(* Schneider Machine Expert - Basic project H_DUSTER, file version 2.9.0.0 *)
(* CompanyInformations: Name=PROMASS, PhoneNumber=+39074238501, Street=Via XXV Aprile, 10/12, City=Trevi, ZipCode=06039, State=PG, Country=Italy, WebSite=www.promass.com *)
(* ProjectInformations: Name=MIXER_EPP, Description=CONTROL TO MIX-UP RECYCLED EPP (EXANDED POLYPROPILENE) WITH FRESH EPP.
AN ADDITIONAL BLOWE IS ADDED TO PERMIT THE OUTPUT FLOW *)
(* UserInformations: LastName=Torroni, FirstName=Stefano, PhoneNumber=+390742385051, Email=info@promass.com, Street=via XXV Aprile, 10/12, City=Trevi, ZipCode=06039, State=Umbria, Country=Italy *)

HARDWARE
  Cpu 0: TM221CE16T
  EthernetConfiguration: NetworkName=M221, IpAllocationMode=FixedAddress, IpAddress=192.168.250.10, SubnetMask=255.255.255.0
  SerialLineConfiguration: Baud=Baud19200, Parity=ParityEven, DataBits=DataBits8, StopBits=StopBits1, PhysicalMedium=PhysicalMediumRs485, TransmissionMode=TransmissionModeIoScannerRtu
  MastTask: UsePeriodScanMode=false, PeriodScan=100
  FastTask: Period=255
  CpuBehavior: StartingMode=StartAutoRunForced, AutoSaveRamOnEeprom=true, WatchdogPeriod=250

SYMBOLS  (address, symbol, comment, settings)
  %M0       DRV_PWR_ON
  %M1       DRV1_JOG_INC
  %M2       DRV1_JOG_DEC
  %M3       DRV2_JOG_INC
  %M4       DRV2_JOG_DEC
  %M5       DRV1_MOVE_VEL
  %M6       DRV2_MOVE_VEL
  %M7       DRV1_ERROR
  %M8       DRV2_ERROR
  %M11      UPP_SENS_ON
  %M12      REM_TANK_FULL_V
  %M13      BLOWER_TOF
  %M20      DRV3_JOG_INC
  %M21      DRV3_JOG_DEC
  %M22      DRV4_JOG_INC
  %M23      DRV4_JOG_DEC
  %M24      DRV3_MOVE_VEL
  %M25      DRV4_MOVE_VEL
  %M26      DRV3_ERROR
  %M27      DRV4_ERROR
  %M30      U1_POWER_ON
  %M31      U2_POWER_ON
  %M32      U3_POWER_ON
  %M33      U4_POWER_ON
  %M34      U1_DRIVE_ERR
  %M35      U2_DRIVE_ERR
  %M36      U3_DRIVE_ERR
  %M37      U4_DRIVE_ERR
  %M40      DRV1_CONTMOTION
  %M41      DRV2_CONTMOTION
  %M42      DRV3_CONTMOTION
  %M43      DRV4_CONTMOTION
  %M100     RATIO_0_CHANGED
  %M101     RATIO_1_CHANGED
  %MW0      DRV1_JOG_SPEED
  %MW1      DRV2_JOG_SPEED
  %MW2      DRV1_MOVEVEL_SPEED
  %MW3      DRV2_MOVE_VEL_SPEED
  %MW4      HMI_ALARMS
  %MW5      FSM
  %MW6      HMI_INP_00  "HMI>>PLC COMMANDS WORD 01"
  %MW7      HMI_OUT_00  "PLC>>HMI FEEDBACK WORD 01"
  %MW8      HMI_OUT_01  "PLC>>HMI FEEDBACK WORD 02"
  %MW9      U1_M1_SPEED_RPM_OUT
  %MW10     U2_M2_SPEED_RPM_OUT
  %MW11     U3_M3_SPEED_RPM_OUT
  %MW12     U4_M4_SPEED_RPM_OUT
  %MW14     DRV3_JOG_SPEED
  %MW15     DRV4_JOG_SPEED
  %MW16     DRV3_MOVEVEL_SPEED
  %MW17     DRV4_MOVEVEL_SPEED
  %MW18     U1_M1_GEARBOX_RATIO  "RECYCLED_MATERIAL SCREW GEARBOX => i=15"
  %MW19     U2_M2_GEARBOX_RATIO  "STAR VALVE INLET GEARBOX => i=120"
  %MW20     U3_M3_GEARBOX_RATIO  "STAR VALVE OUTLET GEARBOX => i=40"
  %MW21     U4_M4_GEARBOX_RATIO  "FAN BLOWER DOES NOT HAVE GEARBOX => i=1"
  %MW22     HMI_INP_02  "HMI>>PLC COMMANDS WORD 02"
  %MW24     HMI_OUT_02  "PLC>>HMI FEEDBACK WORD 03"
  %MW25     FSM_FEEDBACK
  %MW30     DRV1_SPD_AUTO  "RECYCLING MATERIAL DRIVE SPEED AUTOMODE (MULTIPLY BY 2.58 DUE TO GEAR RATIO 12.4/4.8 <=>GEAR_RATIO0/GEAR_RATIO1"
  %MW31     DRV2_SPD_AUTO  "RAW MATERIAL DRIVE SPEED AUTOMODE"
  %MW32     DRV1_SPD_AUTO0
  %MW33     DRV2_SPD_AUTO0
  %MW34     DRV3_SPD_AUTO
  %MW35     DRV4_SPD_AUTO
  %MW36     DRV3_SPD_AUTO0
  %MW37     DRV4_SPD_AUTO0
  %MC_JOG_ATV0   [Axis(Value(DriveAxis=DRV0)), Vel(Value(short=210))]
  %MC_JOG_ATV1   [Axis(Value(DriveAxis=DRV1)), Vel(Value(short=210))]
  %MC_JOG_ATV2   [Axis(Value(DriveAxis=DRV2)), Vel(Value(short=210))]
  %MC_JOG_ATV3   [Axis(Value(DriveAxis=DRV3)), Vel(Value(short=400))]
  %MC_MOVEVEL_ATV0   [Axis(Value(DriveAxis=DRV0)), Vel(Value(short=0))]
  %MC_MOVEVEL_ATV1   [Axis(Value(DriveAxis=DRV1)), Vel(Value(short=0))]
  %MC_MOVEVEL_ATV2   [Axis(Value(DriveAxis=DRV2)), Vel(Value(short=0))]
  %MC_MOVEVEL_ATV3   [Axis(Value(DriveAxis=DRV3)), Vel(Value(short=0))]
  %MC_POWER_ATV0   [Axis(Value(DriveAxis=DRV0))]
  %MC_POWER_ATV1   [Axis(Value(DriveAxis=DRV1))]
  %MC_POWER_ATV2   [Axis(Value(DriveAxis=DRV2))]
  %MC_POWER_ATV3   [Axis(Value(DriveAxis=DRV3))]
  %MC_READMOTIONSTATE_ATV0   [Axis(Value(DriveAxis=DRV0))]
  %MC_READMOTIONSTATE_ATV1   [Axis(Value(DriveAxis=DRV1))]
  %MC_READMOTIONSTATE_ATV2   [Axis(Value(DriveAxis=DRV2))]
  %MC_READMOTIONSTATE_ATV3   [Axis(Value(DriveAxis=DRV3))]
  %MC_READSTATUS_ATV0   [Axis(Value(DriveAxis=DRV0))]
  %MC_READSTATUS_ATV1   [Axis(Value(DriveAxis=DRV1))]
  %MC_READSTATUS_ATV2   [Axis(Value(DriveAxis=DRV2))]
  %MC_READSTATUS_ATV3   [Axis(Value(DriveAxis=DRV3))]
  %MC_RESET_ATV0   [Axis(Value(DriveAxis=DRV0))]
  %MC_RESET_ATV1   [Axis(Value(DriveAxis=DRV1))]
  %MC_RESET_ATV2   [Axis(Value(DriveAxis=DRV2))]
  %MC_RESET_ATV3   [Axis(Value(DriveAxis=DRV3))]
  %MC_STOP_ATV0   [Axis(Value(DriveAxis=DRV0))]
  %MC_STOP_ATV1   [Axis(Value(DriveAxis=DRV1))]
  %MC_STOP_ATV2   [Axis(Value(DriveAxis=DRV2))]
  %MC_STOP_ATV3   [Axis(Value(DriveAxis=DRV3))]
  %I0.0     START_BTN
  %I0.1     STOP_BTN
  %I0.2     QM1
  %I0.3     QM2
  %I0.4     QM3
  %I0.5     QM4
  %Q0.0     STO
  %Q0.1     KA2_MILL_01_IF
  %Q0.2     KA3_MILL_02_IF

POU MAIN
  (* SectionNumber=1 *)

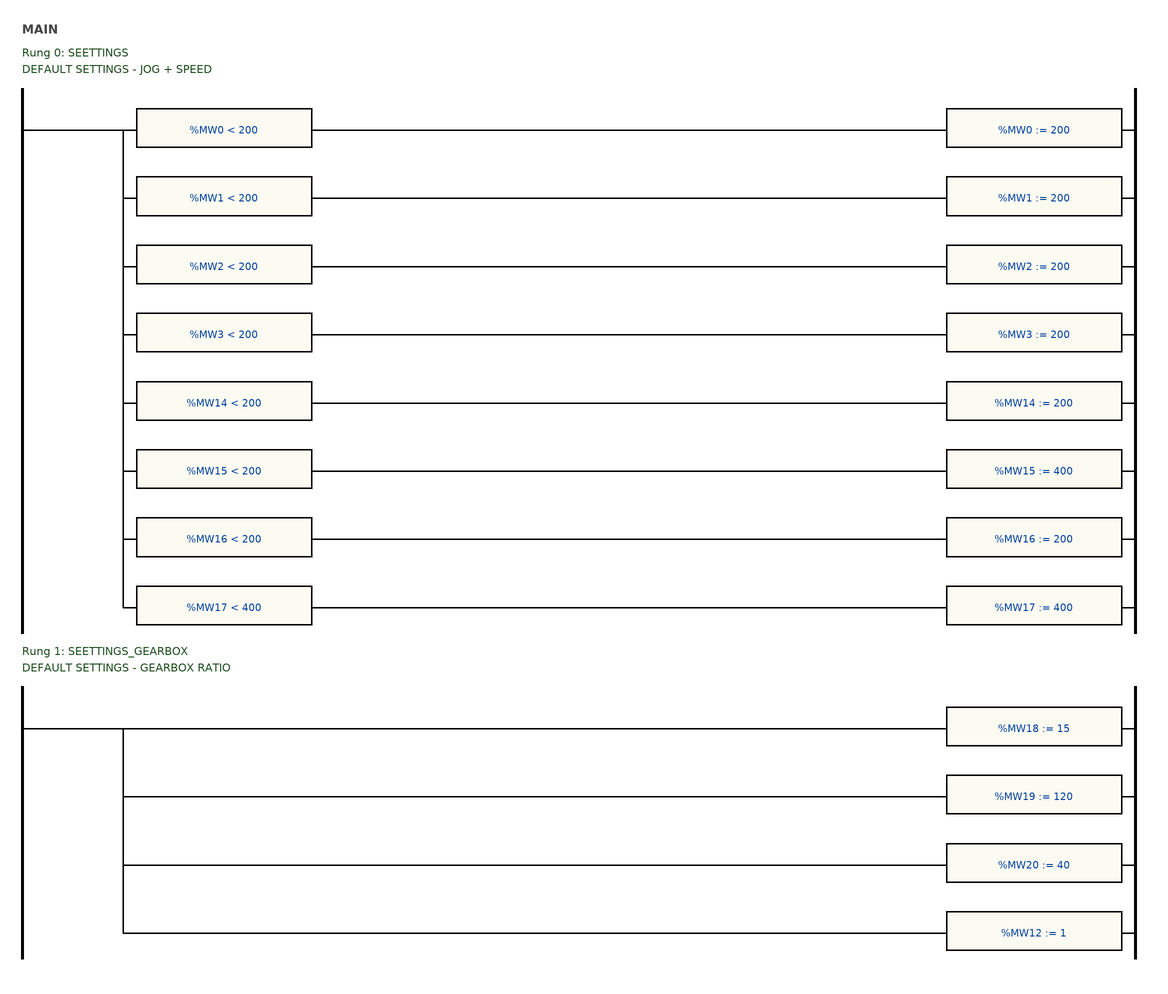

// Rung 0: SEETTINGS
// DEFAULT SETTINGS - JOG + SPEED
  LD 1
  MPS
  AND [ %MW0 < 200 ]      (* DRV1_JOG_SPEED *)
  [ %MW0 := 200 ]         (* DRV1_JOG_SPEED *)
  MRD
  AND [ %MW1 < 200 ]      (* DRV2_JOG_SPEED *)
  [ %MW1 := 200 ]         (* DRV2_JOG_SPEED *)
  MRD
  AND [ %MW2 < 200 ]      (* DRV1_MOVEVEL_SPEED *)
  [ %MW2 := 200 ]         (* DRV1_MOVEVEL_SPEED *)
  MRD
  AND [ %MW3 < 200 ]      (* DRV2_MOVE_VEL_SPEED *)
  [ %MW3 := 200 ]         (* DRV2_MOVE_VEL_SPEED *)
  MRD
  AND [ %MW14 < 200 ]     (* DRV3_JOG_SPEED *)
  [ %MW14 := 200 ]        (* DRV3_JOG_SPEED *)
  MRD
  AND [ %MW15 < 200 ]     (* DRV4_JOG_SPEED *)
  [ %MW15 := 400 ]        (* DRV4_JOG_SPEED *)
  MRD
  AND [ %MW16 < 200 ]     (* DRV3_MOVEVEL_SPEED *)
  [ %MW16 := 200 ]        (* DRV3_MOVEVEL_SPEED *)
  MPP
  AND [ %MW17 < 400 ]     (* DRV4_MOVEVEL_SPEED *)
  [ %MW17 := 400 ]        (* DRV4_MOVEVEL_SPEED *)
  // as ST:
  //   IF DRV1_JOG_SPEED < 200 THEN DRV1_JOG_SPEED := 200; END_IF;
  //   IF DRV2_JOG_SPEED < 200 THEN DRV2_JOG_SPEED := 200; END_IF;
  //   IF DRV1_MOVEVEL_SPEED < 200 THEN DRV1_MOVEVEL_SPEED := 200; END_IF;
  //   IF DRV2_MOVE_VEL_SPEED < 200 THEN DRV2_MOVE_VEL_SPEED := 200; END_IF;
  //   IF DRV3_JOG_SPEED < 200 THEN DRV3_JOG_SPEED := 200; END_IF;
  //   IF DRV4_JOG_SPEED < 200 THEN DRV4_JOG_SPEED := 400; END_IF;
  //   IF DRV3_MOVEVEL_SPEED < 200 THEN DRV3_MOVEVEL_SPEED := 200; END_IF;
  //   IF DRV4_MOVEVEL_SPEED < 400 THEN DRV4_MOVEVEL_SPEED := 400; END_IF;

// Rung 1: SEETTINGS_GEARBOX
// DEFAULT SETTINGS - GEARBOX RATIO
  LD 1
  [ %MW18 := 15 ]         (* U1_M1_GEARBOX_RATIO *)
  [ %MW19 := 120 ]        (* U2_M2_GEARBOX_RATIO *)
  [ %MW20 := 40 ]         (* U3_M3_GEARBOX_RATIO *)
  [ %MW12 := 1 ]          (* U4_M4_SPEED_RPM_OUT *)
  // as ST:
  //   U1_M1_GEARBOX_RATIO := 15;
  //   U2_M2_GEARBOX_RATIO := 120;
  //   U3_M3_GEARBOX_RATIO := 40;
  //   U4_M4_SPEED_RPM_OUT := 1;

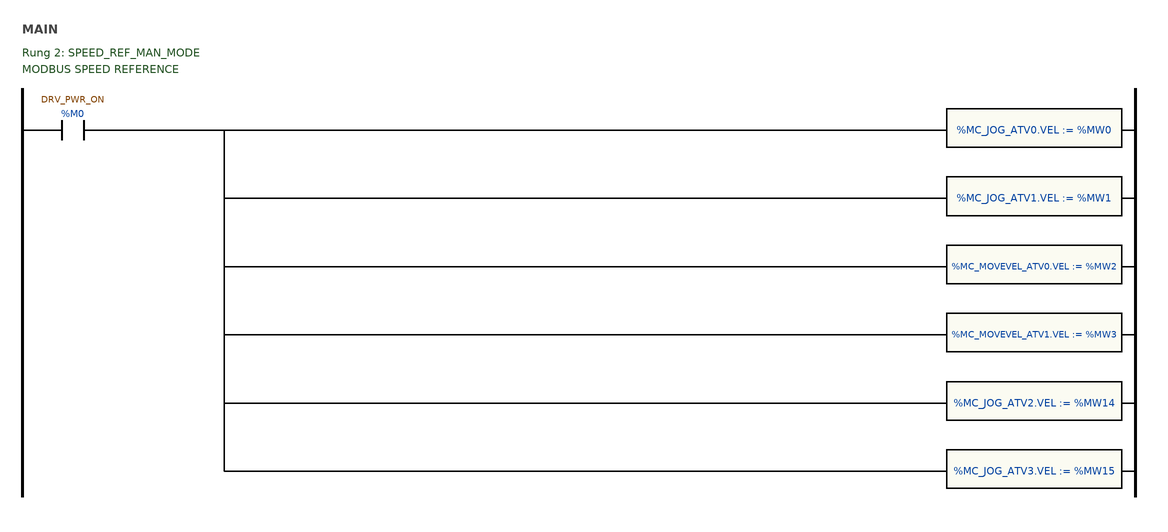

// Rung 2: SPEED_REF_MAN_MODE
// MODBUS SPEED REFERENCE
  LD %M0                  (* DRV_PWR_ON *)
  [ %MC_JOG_ATV0.VEL := %MW0 ](* DRV1_JOG_SPEED *)
  [ %MC_JOG_ATV1.VEL := %MW1 ](* DRV2_JOG_SPEED *)
  [ %MC_MOVEVEL_ATV0.VEL := %MW2 ](* DRV1_MOVEVEL_SPEED *)
  [ %MC_MOVEVEL_ATV1.VEL := %MW3 ](* DRV2_MOVE_VEL_SPEED *)
  [ %MC_JOG_ATV2.VEL := %MW14 ](* DRV3_JOG_SPEED *)
  [ %MC_JOG_ATV3.VEL := %MW15 ](* DRV4_JOG_SPEED *)
  // as ST:
  //   IF DRV_PWR_ON THEN %MC_JOG_ATV0.VEL := DRV1_JOG_SPEED; END_IF;
  //   IF DRV_PWR_ON THEN %MC_JOG_ATV1.VEL := DRV2_JOG_SPEED; END_IF;
  //   IF DRV_PWR_ON THEN %MC_MOVEVEL_ATV0.VEL := DRV1_MOVEVEL_SPEED; END_IF;
  //   IF DRV_PWR_ON THEN %MC_MOVEVEL_ATV1.VEL := DRV2_MOVE_VEL_SPEED; END_IF;
  //   IF DRV_PWR_ON THEN %MC_JOG_ATV2.VEL := DRV3_JOG_SPEED; END_IF;
  //   IF DRV_PWR_ON THEN %MC_JOG_ATV3.VEL := DRV4_JOG_SPEED; END_IF;

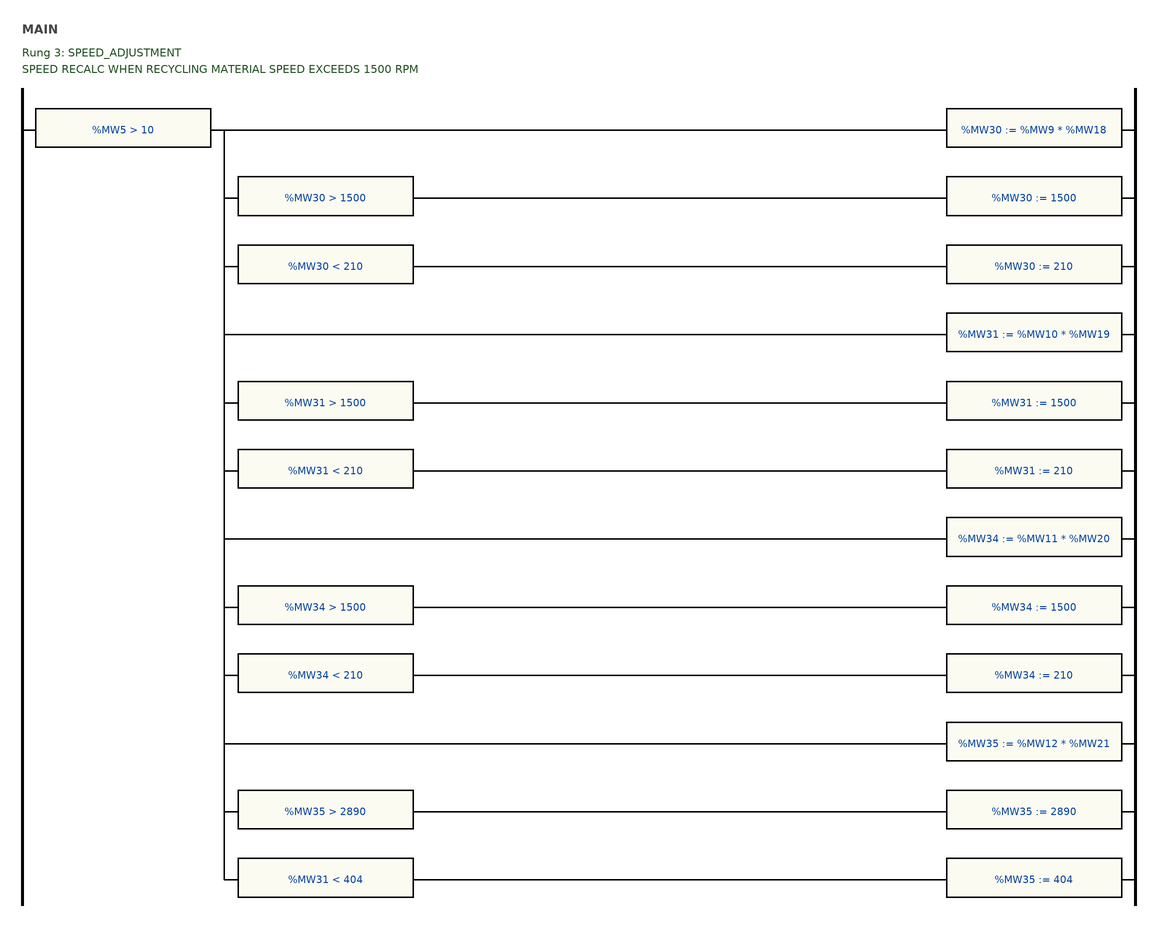

// Rung 3: SPEED_ADJUSTMENT
// SPEED RECALC WHEN RECYCLING MATERIAL SPEED EXCEEDS 1500 RPM
  LD [ %MW5 > 10 ]        (* FSM *)
  MPS
  [ %MW30 := %MW9 * %MW18 ](* DRV1_SPD_AUTO, U1_M1_SPEED_RPM_OUT, U1_M1_GEARBOX_RATIO *)
  MRD
  AND [ %MW30 > 1500 ]    (* DRV1_SPD_AUTO *)
  [ %MW30 := 1500 ]       (* DRV1_SPD_AUTO *)
  MRD
  AND [ %MW30 < 210 ]     (* DRV1_SPD_AUTO *)
  [ %MW30 := 210 ]        (* DRV1_SPD_AUTO *)
  MRD
  [ %MW31 := %MW10 * %MW19 ](* DRV2_SPD_AUTO, U2_M2_SPEED_RPM_OUT, U2_M2_GEARBOX_RATIO *)
  MRD
  AND [ %MW31 > 1500 ]    (* DRV2_SPD_AUTO *)
  [ %MW31 := 1500 ]       (* DRV2_SPD_AUTO *)
  MRD
  AND [ %MW31 < 210 ]     (* DRV2_SPD_AUTO *)
  [ %MW31 := 210 ]        (* DRV2_SPD_AUTO *)
  MRD
  [ %MW34 := %MW11 * %MW20 ](* DRV3_SPD_AUTO, U3_M3_SPEED_RPM_OUT, U3_M3_GEARBOX_RATIO *)
  MRD
  AND [ %MW34 > 1500 ]    (* DRV3_SPD_AUTO *)
  [ %MW34 := 1500 ]       (* DRV3_SPD_AUTO *)
  MRD
  AND [ %MW34 < 210 ]     (* DRV3_SPD_AUTO *)
  [ %MW34 := 210 ]        (* DRV3_SPD_AUTO *)
  MRD
  [ %MW35 := %MW12 * %MW21 ](* DRV4_SPD_AUTO, U4_M4_SPEED_RPM_OUT, U4_M4_GEARBOX_RATIO *)
  MRD
  AND [ %MW35 > 2890 ]    (* DRV4_SPD_AUTO *)
  [ %MW35 := 2890 ]       (* DRV4_SPD_AUTO *)
  MPP
  AND [ %MW31 < 404 ]     (* DRV2_SPD_AUTO *)
  [ %MW35 := 404 ]        (* DRV4_SPD_AUTO *)
  // as ST:
  //   IF FSM > 10 THEN DRV1_SPD_AUTO := U1_M1_SPEED_RPM_OUT * U1_M1_GEARBOX_RATIO; END_IF;
  //   IF FSM > 10 AND DRV1_SPD_AUTO > 1500 THEN DRV1_SPD_AUTO := 1500; END_IF;
  //   IF FSM > 10 AND DRV1_SPD_AUTO < 210 THEN DRV1_SPD_AUTO := 210; END_IF;
  //   IF FSM > 10 THEN DRV2_SPD_AUTO := U2_M2_SPEED_RPM_OUT * U2_M2_GEARBOX_RATIO; END_IF;
  //   IF FSM > 10 AND DRV2_SPD_AUTO > 1500 THEN DRV2_SPD_AUTO := 1500; END_IF;
  //   IF FSM > 10 AND DRV2_SPD_AUTO < 210 THEN DRV2_SPD_AUTO := 210; END_IF;
  //   IF FSM > 10 THEN DRV3_SPD_AUTO := U3_M3_SPEED_RPM_OUT * U3_M3_GEARBOX_RATIO; END_IF;
  //   IF FSM > 10 AND DRV3_SPD_AUTO > 1500 THEN DRV3_SPD_AUTO := 1500; END_IF;
  //   IF FSM > 10 AND DRV3_SPD_AUTO < 210 THEN DRV3_SPD_AUTO := 210; END_IF;
  //   IF FSM > 10 THEN DRV4_SPD_AUTO := U4_M4_SPEED_RPM_OUT * U4_M4_GEARBOX_RATIO; END_IF;
  //   IF FSM > 10 AND DRV4_SPD_AUTO > 2890 THEN DRV4_SPD_AUTO := 2890; END_IF;
  //   IF FSM > 10 AND DRV2_SPD_AUTO < 404 THEN DRV4_SPD_AUTO := 404; END_IF;

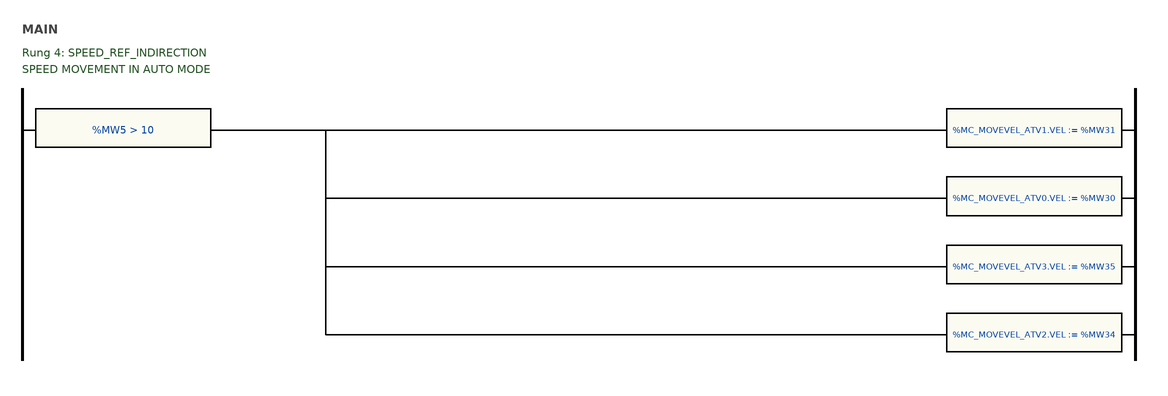

// Rung 4: SPEED_REF_INDIRECTION
// SPEED MOVEMENT IN AUTO MODE
  LD [ %MW5 > 10 ]        (* FSM *)
  [ %MC_MOVEVEL_ATV1.VEL := %MW31 ](* DRV2_SPD_AUTO *)
  [ %MC_MOVEVEL_ATV0.VEL := %MW30 ](* DRV1_SPD_AUTO *)
  [ %MC_MOVEVEL_ATV3.VEL := %MW35 ](* DRV4_SPD_AUTO *)
  [ %MC_MOVEVEL_ATV2.VEL := %MW34 ](* DRV3_SPD_AUTO *)
  // as ST:
  //   IF FSM > 10 THEN %MC_MOVEVEL_ATV1.VEL := DRV2_SPD_AUTO; END_IF;
  //   IF FSM > 10 THEN %MC_MOVEVEL_ATV0.VEL := DRV1_SPD_AUTO; END_IF;
  //   IF FSM > 10 THEN %MC_MOVEVEL_ATV3.VEL := DRV4_SPD_AUTO; END_IF;
  //   IF FSM > 10 THEN %MC_MOVEVEL_ATV2.VEL := DRV3_SPD_AUTO; END_IF;

POU FSM+CMD+HMI
  (* SectionNumber=2 *)

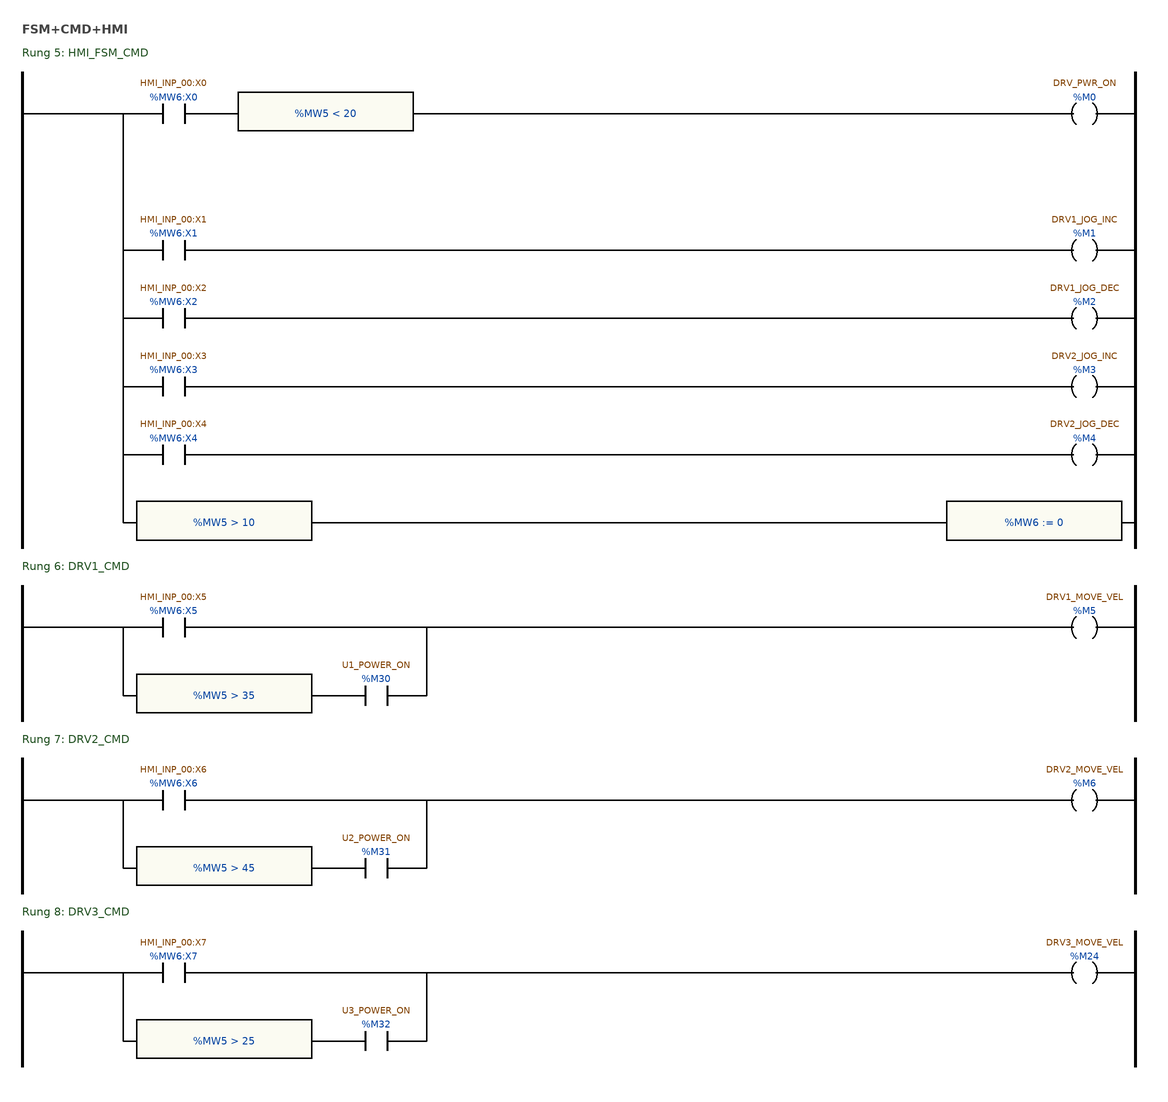

// Rung 5: HMI_FSM_CMD
  LD 1
  MPS
  AND %MW6:X0             (* HMI_INP_00 *)
  AND [ %MW5 < 20 ]       (* FSM *)
  ST %M0                  (* DRV_PWR_ON *)
  MRD
  AND %MW6:X1             (* HMI_INP_00 *)
  ST %M1                  (* DRV1_JOG_INC *)
  MRD
  AND %MW6:X2             (* HMI_INP_00 *)
  ST %M2                  (* DRV1_JOG_DEC *)
  MRD
  AND %MW6:X3             (* HMI_INP_00 *)
  ST %M3                  (* DRV2_JOG_INC *)
  MRD
  AND %MW6:X4             (* HMI_INP_00 *)
  ST %M4                  (* DRV2_JOG_DEC *)
  MPP
  AND [ %MW5 > 10 ]       (* FSM *)
  [ %MW6 := 0 ]           (* HMI_INP_00 *)
  // as ST:
  //   DRV_PWR_ON := HMI_INP_00:X0 AND FSM < 20;
  //   DRV1_JOG_INC := HMI_INP_00:X1;
  //   DRV1_JOG_DEC := HMI_INP_00:X2;
  //   DRV2_JOG_INC := HMI_INP_00:X3;
  //   DRV2_JOG_DEC := HMI_INP_00:X4;
  //   IF FSM > 10 THEN HMI_INP_00 := 0; END_IF;

// Rung 6: DRV1_CMD
  LD 1
  AND( %MW6:X5            (* HMI_INP_00 *)
  OR( [ %MW5 > 35 ]       (* FSM *)
  AND %M30                (* U1_POWER_ON *)
  )
  )
  ST %M5                  (* DRV1_MOVE_VEL *)
  // as ST:
  //   DRV1_MOVE_VEL := HMI_INP_00:X5 OR FSM > 35 AND U1_POWER_ON;

// Rung 7: DRV2_CMD
  LD 1
  AND( %MW6:X6            (* HMI_INP_00 *)
  OR( [ %MW5 > 45 ]       (* FSM *)
  AND %M31                (* U2_POWER_ON *)
  )
  )
  ST %M6                  (* DRV2_MOVE_VEL *)
  // as ST:
  //   DRV2_MOVE_VEL := HMI_INP_00:X6 OR FSM > 45 AND U2_POWER_ON;

// Rung 8: DRV3_CMD
  LD 1
  AND( %MW6:X7            (* HMI_INP_00 *)
  OR( [ %MW5 > 25 ]       (* FSM *)
  AND %M32                (* U3_POWER_ON *)
  )
  )
  ST %M24                 (* DRV3_MOVE_VEL *)
  // as ST:
  //   DRV3_MOVE_VEL := HMI_INP_00:X7 OR FSM > 25 AND U3_POWER_ON;

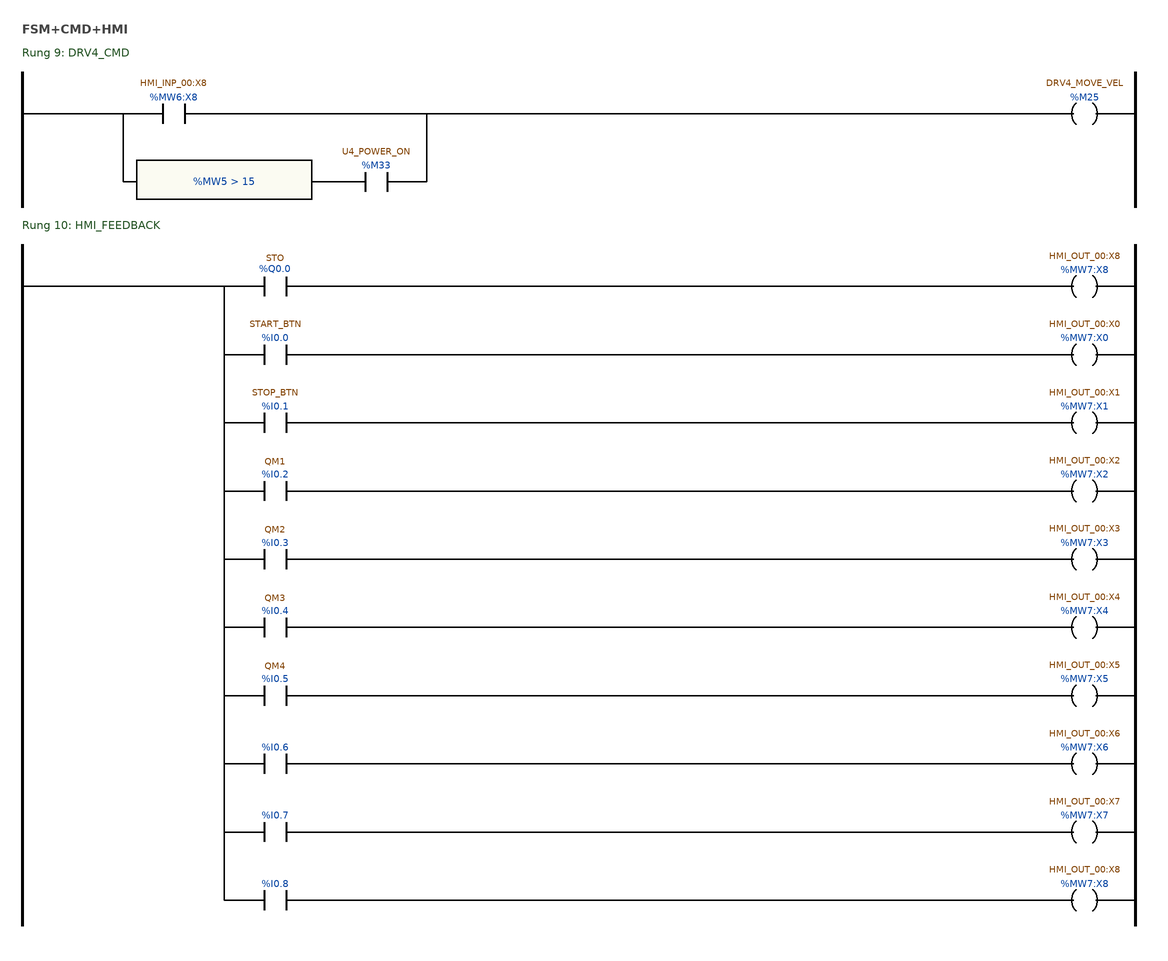

// Rung 9: DRV4_CMD
  LD 1
  AND( %MW6:X8            (* HMI_INP_00 *)
  OR( [ %MW5 > 15 ]       (* FSM *)
  AND %M33                (* U4_POWER_ON *)
  )
  )
  ST %M25                 (* DRV4_MOVE_VEL *)
  // as ST:
  //   DRV4_MOVE_VEL := HMI_INP_00:X8 OR FSM > 15 AND U4_POWER_ON;

// Rung 10: HMI_FEEDBACK
  LD 1
  MPS
  AND %Q0.0               (* STO *)
  ST %MW7:X8              (* HMI_OUT_00 *)
  MRD
  AND %I0.0               (* START_BTN *)
  ST %MW7:X0              (* HMI_OUT_00 *)
  MRD
  AND %I0.1               (* STOP_BTN *)
  ST %MW7:X1              (* HMI_OUT_00 *)
  MRD
  AND %I0.2               (* QM1 *)
  ST %MW7:X2              (* HMI_OUT_00 *)
  MRD
  AND %I0.3               (* QM2 *)
  ST %MW7:X3              (* HMI_OUT_00 *)
  MRD
  AND %I0.4               (* QM3 *)
  ST %MW7:X4              (* HMI_OUT_00 *)
  MRD
  AND %I0.5               (* QM4 *)
  ST %MW7:X5              (* HMI_OUT_00 *)
  MRD
  AND %I0.6
  ST %MW7:X6              (* HMI_OUT_00 *)
  MRD
  AND %I0.7
  ST %MW7:X7              (* HMI_OUT_00 *)
  MPP
  AND %I0.8
  ST %MW7:X8              (* HMI_OUT_00 *)
  // as ST:
  //   HMI_OUT_00:X8 := STO;
  //   HMI_OUT_00:X0 := START_BTN;
  //   HMI_OUT_00:X1 := STOP_BTN;
  //   HMI_OUT_00:X2 := QM1;
  //   HMI_OUT_00:X3 := QM2;
  //   HMI_OUT_00:X4 := QM3;
  //   HMI_OUT_00:X5 := QM4;
  //   HMI_OUT_00:X6 := %I0.6;
  //   HMI_OUT_00:X7 := %I0.7;
  //   HMI_OUT_00:X8 := %I0.8;

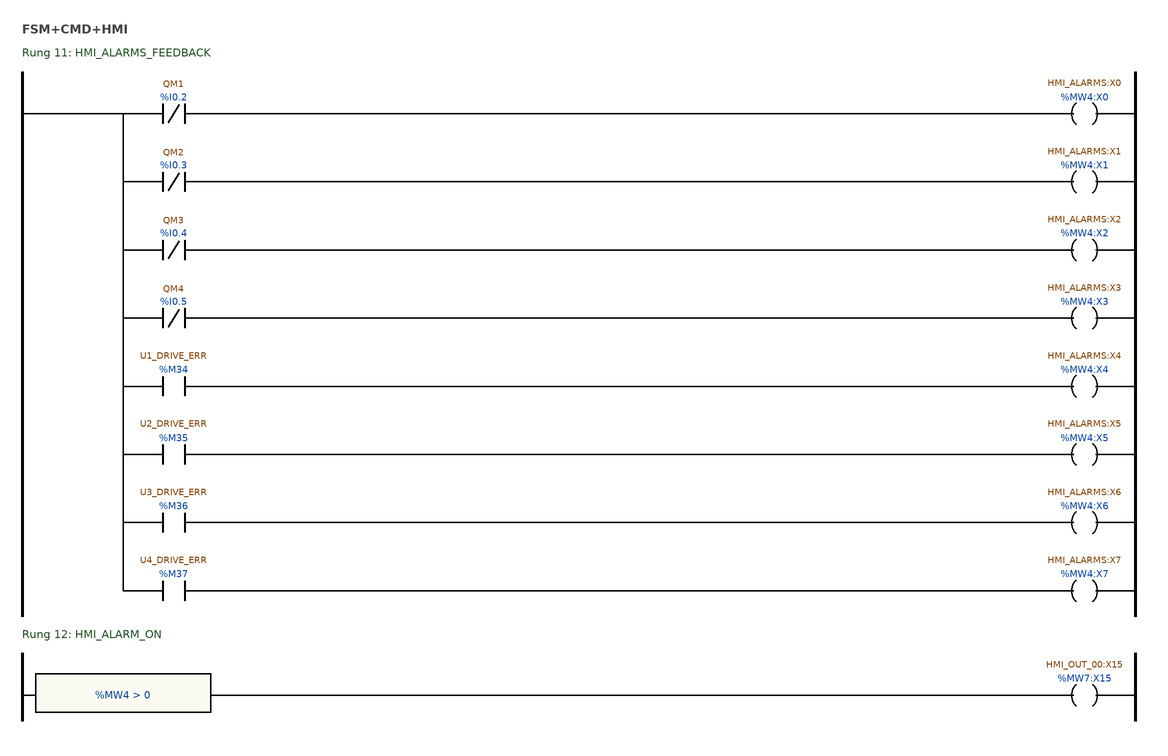

// Rung 11: HMI_ALARMS_FEEDBACK
  LD 1
  MPS
  ANDN %I0.2              (* QM1 *)
  ST %MW4:X0              (* HMI_ALARMS *)
  MRD
  ANDN %I0.3              (* QM2 *)
  ST %MW4:X1              (* HMI_ALARMS *)
  MRD
  ANDN %I0.4              (* QM3 *)
  ST %MW4:X2              (* HMI_ALARMS *)
  MRD
  ANDN %I0.5              (* QM4 *)
  ST %MW4:X3              (* HMI_ALARMS *)
  MRD
  AND %M34                (* U1_DRIVE_ERR *)
  ST %MW4:X4              (* HMI_ALARMS *)
  MRD
  AND %M35                (* U2_DRIVE_ERR *)
  ST %MW4:X5              (* HMI_ALARMS *)
  MRD
  AND %M36                (* U3_DRIVE_ERR *)
  ST %MW4:X6              (* HMI_ALARMS *)
  MPP
  AND %M37                (* U4_DRIVE_ERR *)
  ST %MW4:X7              (* HMI_ALARMS *)
  // as ST:
  //   HMI_ALARMS:X0 := NOT QM1;
  //   HMI_ALARMS:X1 := NOT QM2;
  //   HMI_ALARMS:X2 := NOT QM3;
  //   HMI_ALARMS:X3 := NOT QM4;
  //   HMI_ALARMS:X4 := U1_DRIVE_ERR;
  //   HMI_ALARMS:X5 := U2_DRIVE_ERR;
  //   HMI_ALARMS:X6 := U3_DRIVE_ERR;
  //   HMI_ALARMS:X7 := U4_DRIVE_ERR;

// Rung 12: HMI_ALARM_ON
  LD [ %MW4 > 0 ]         (* HMI_ALARMS *)
  ST %MW7:X15             (* HMI_OUT_00 *)
  // as ST:
  //   HMI_OUT_00:X15 := HMI_ALARMS > 0;

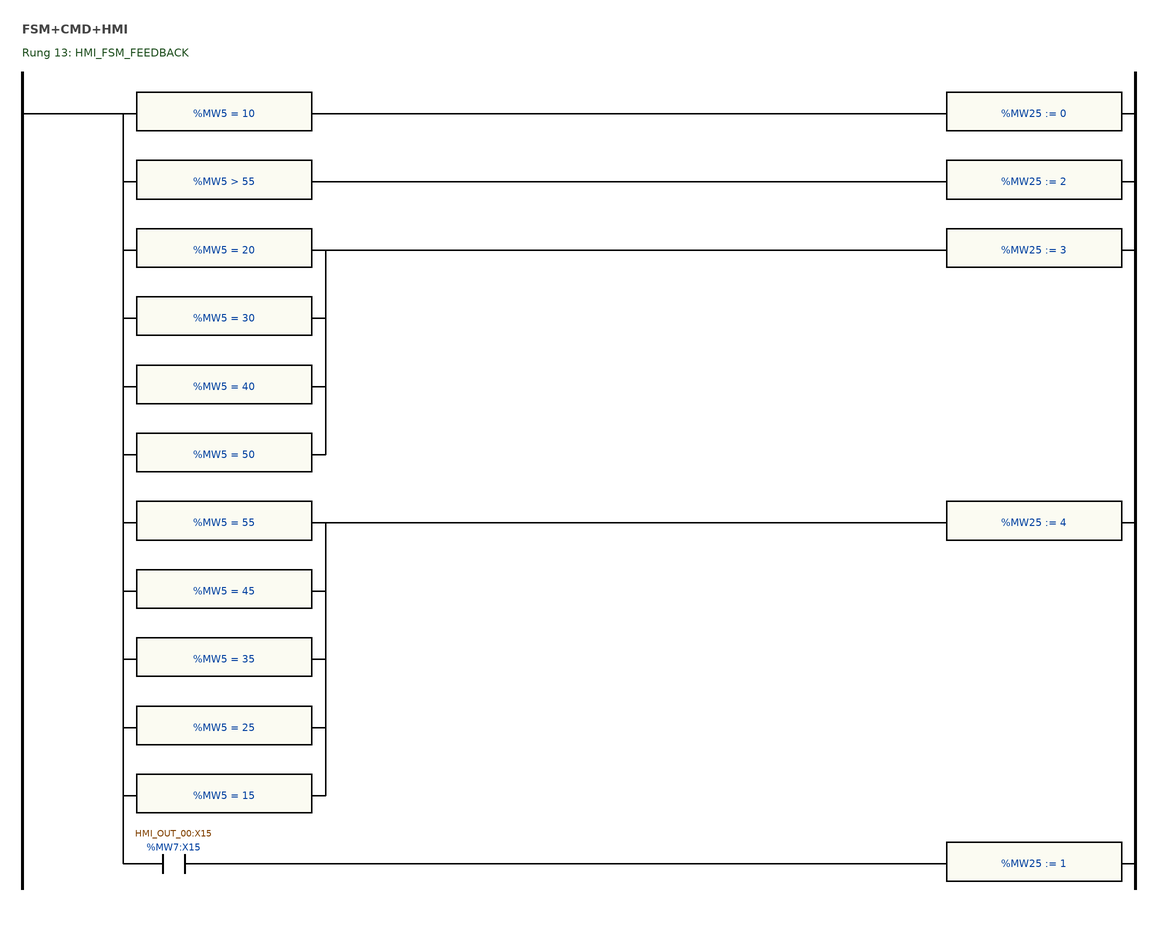

// Rung 13: HMI_FSM_FEEDBACK
  LD 1
  MPS
  AND [ %MW5 = 10 ]       (* FSM *)
  [ %MW25 := 0 ]          (* FSM_FEEDBACK *)
  MRD
  AND [ %MW5 > 55 ]       (* FSM *)
  [ %MW25 := 2 ]          (* FSM_FEEDBACK *)
  MRD
  AND( [ %MW5 = 20 ]      (* FSM *)
  OR [ %MW5 = 30 ]        (* FSM *)
  OR [ %MW5 = 40 ]        (* FSM *)
  OR [ %MW5 = 50 ]        (* FSM *)
  )
  [ %MW25 := 3 ]          (* FSM_FEEDBACK *)
  MRD
  AND( [ %MW5 = 55 ]      (* FSM *)
  OR [ %MW5 = 45 ]        (* FSM *)
  OR [ %MW5 = 35 ]        (* FSM *)
  OR [ %MW5 = 25 ]        (* FSM *)
  OR [ %MW5 = 15 ]        (* FSM *)
  )
  [ %MW25 := 4 ]          (* FSM_FEEDBACK *)
  MPP
  AND %MW7:X15            (* HMI_OUT_00 *)
  [ %MW25 := 1 ]          (* FSM_FEEDBACK *)
  // as ST:
  //   IF FSM = 10 THEN FSM_FEEDBACK := 0; END_IF;
  //   IF FSM > 55 THEN FSM_FEEDBACK := 2; END_IF;
  //   IF FSM = 20 OR FSM = 30 OR FSM = 40 OR FSM = 50 THEN FSM_FEEDBACK := 3; END_IF;
  //   IF FSM = 55 OR FSM = 45 OR FSM = 35 OR FSM = 25 OR FSM = 15 THEN FSM_FEEDBACK := 4; END_IF;
  //   IF HMI_OUT_00:X15 THEN FSM_FEEDBACK := 1; END_IF;

POU FSM
  (* SectionNumber=3 *)

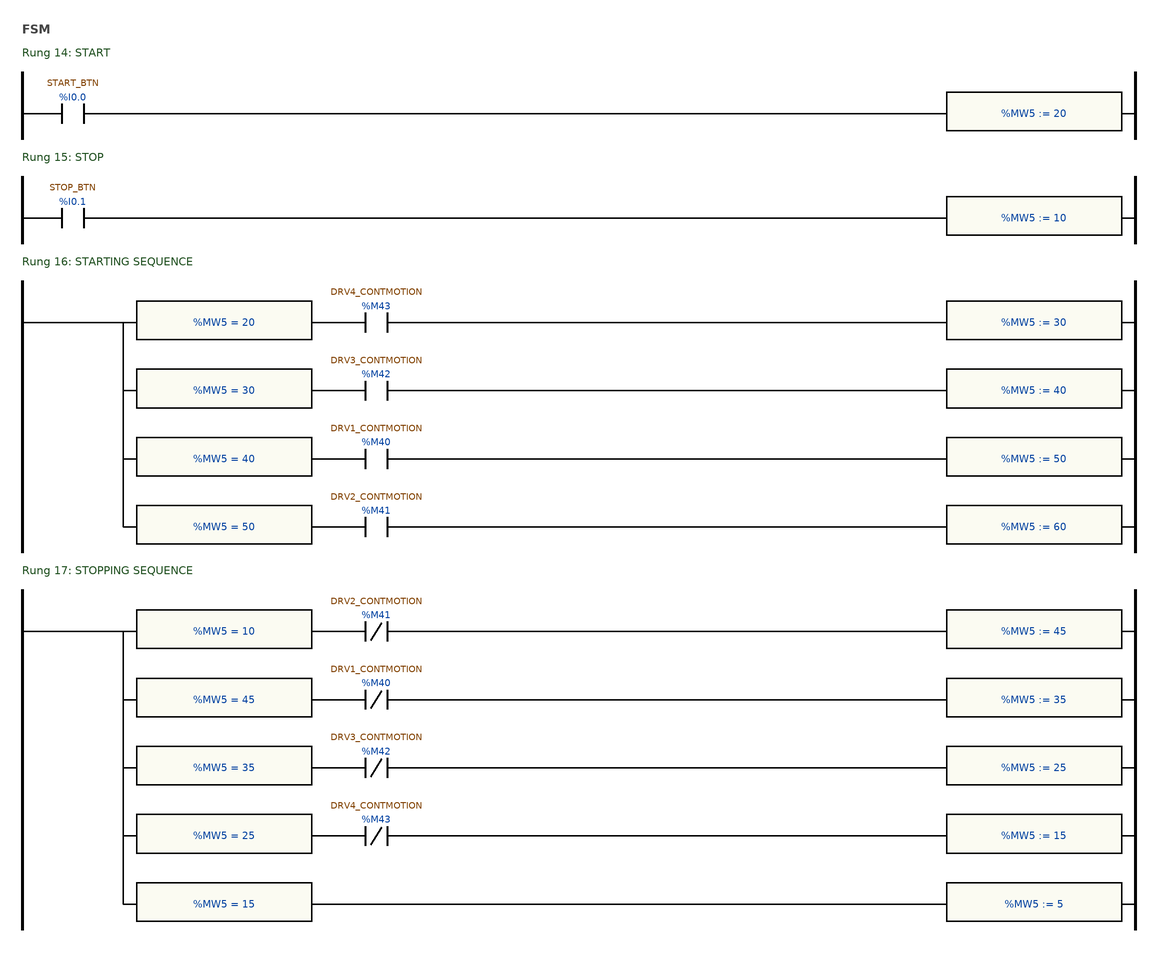

// Rung 14: START
  LD %I0.0                (* START_BTN *)
  [ %MW5 := 20 ]          (* FSM *)
  // as ST:
  //   IF START_BTN THEN FSM := 20; END_IF;

// Rung 15: STOP
  LD %I0.1                (* STOP_BTN *)
  [ %MW5 := 10 ]          (* FSM *)
  // as ST:
  //   IF STOP_BTN THEN FSM := 10; END_IF;

// Rung 16: STARTING SEQUENCE
  LD 1
  MPS
  AND [ %MW5 = 20 ]       (* FSM *)
  AND %M43                (* DRV4_CONTMOTION *)
  [ %MW5 := 30 ]          (* FSM *)
  MRD
  AND [ %MW5 = 30 ]       (* FSM *)
  AND %M42                (* DRV3_CONTMOTION *)
  [ %MW5 := 40 ]          (* FSM *)
  MRD
  AND [ %MW5 = 40 ]       (* FSM *)
  AND %M40                (* DRV1_CONTMOTION *)
  [ %MW5 := 50 ]          (* FSM *)
  MPP
  AND [ %MW5 = 50 ]       (* FSM *)
  AND %M41                (* DRV2_CONTMOTION *)
  [ %MW5 := 60 ]          (* FSM *)
  // as ST:
  //   IF FSM = 20 AND DRV4_CONTMOTION THEN FSM := 30; END_IF;
  //   IF FSM = 30 AND DRV3_CONTMOTION THEN FSM := 40; END_IF;
  //   IF FSM = 40 AND DRV1_CONTMOTION THEN FSM := 50; END_IF;
  //   IF FSM = 50 AND DRV2_CONTMOTION THEN FSM := 60; END_IF;

// Rung 17: STOPPING SEQUENCE
  LD 1
  MPS
  AND [ %MW5 = 10 ]       (* FSM *)
  ANDN %M41               (* DRV2_CONTMOTION *)
  [ %MW5 := 45 ]          (* FSM *)
  MRD
  AND [ %MW5 = 45 ]       (* FSM *)
  ANDN %M40               (* DRV1_CONTMOTION *)
  [ %MW5 := 35 ]          (* FSM *)
  MRD
  AND [ %MW5 = 35 ]       (* FSM *)
  ANDN %M42               (* DRV3_CONTMOTION *)
  [ %MW5 := 25 ]          (* FSM *)
  MRD
  AND [ %MW5 = 25 ]       (* FSM *)
  ANDN %M43               (* DRV4_CONTMOTION *)
  [ %MW5 := 15 ]          (* FSM *)
  MPP
  AND [ %MW5 = 15 ]       (* FSM *)
  [ %MW5 := 5 ]           (* FSM *)
  // as ST:
  //   IF FSM = 10 AND NOT DRV2_CONTMOTION THEN FSM := 45; END_IF;
  //   IF FSM = 45 AND NOT DRV1_CONTMOTION THEN FSM := 35; END_IF;
  //   IF FSM = 35 AND NOT DRV3_CONTMOTION THEN FSM := 25; END_IF;
  //   IF FSM = 25 AND NOT DRV4_CONTMOTION THEN FSM := 15; END_IF;
  //   IF FSM = 15 THEN FSM := 5; END_IF;

POU OUT
  (* SectionNumber=5 *)

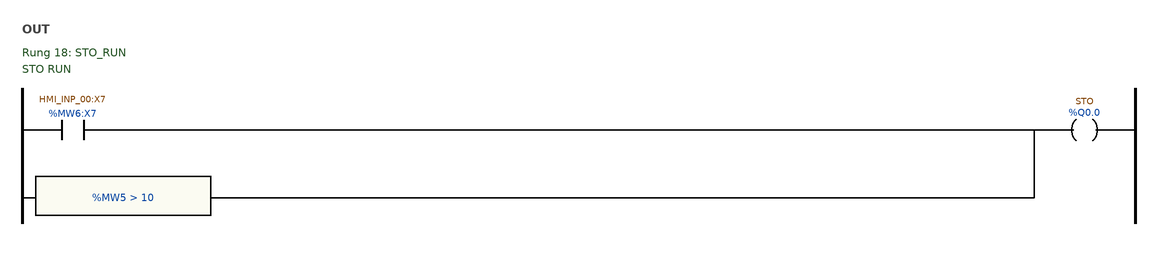

// Rung 18: STO_RUN
// STO RUN
  LD %MW6:X7              (* HMI_INP_00 *)
  OR [ %MW5 > 10 ]        (* FSM *)
  ST %Q0.0                (* STO *)
  // as ST:
  //   STO := HMI_INP_00:X7 OR FSM > 10;

POU DRIVE_JOG
  (* SectionNumber=0 *)

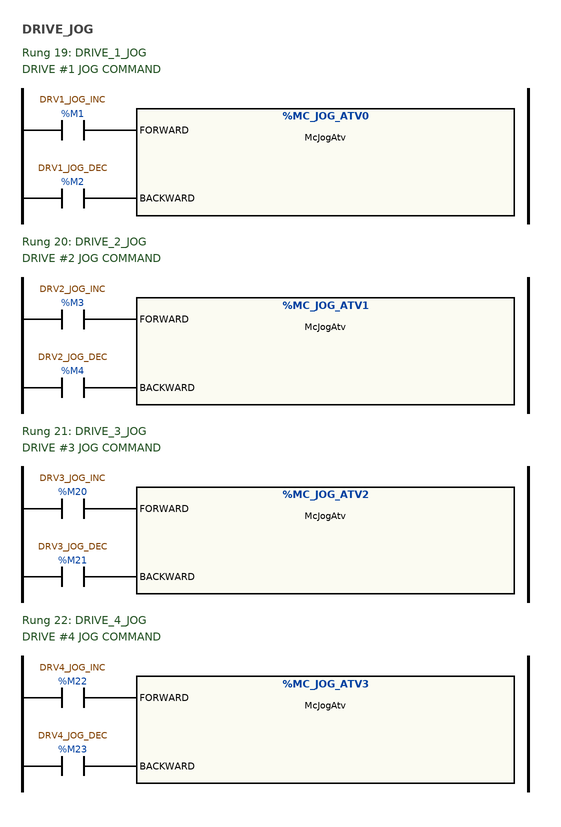

// Rung 19: DRIVE_1_JOG
// DRIVE #1 JOG COMMAND
  BLK %MC_JOG_ATV0
  LD %M1                  (* DRV1_JOG_INC *)
  FORWARD
  LD %M2                  (* DRV1_JOG_DEC *)
  BACKWARD
  END_BLK
  // as ST:
  //   %MC_JOG_ATV0(FORWARD := DRV1_JOG_INC, BACKWARD := DRV1_JOG_DEC);

// Rung 20: DRIVE_2_JOG
// DRIVE #2 JOG COMMAND
  BLK %MC_JOG_ATV1
  LD %M3                  (* DRV2_JOG_INC *)
  FORWARD
  LD %M4                  (* DRV2_JOG_DEC *)
  BACKWARD
  END_BLK
  // as ST:
  //   %MC_JOG_ATV1(FORWARD := DRV2_JOG_INC, BACKWARD := DRV2_JOG_DEC);

// Rung 21: DRIVE_3_JOG
// DRIVE #3 JOG COMMAND
  BLK %MC_JOG_ATV2
  LD %M20                 (* DRV3_JOG_INC *)
  FORWARD
  LD %M21                 (* DRV3_JOG_DEC *)
  BACKWARD
  END_BLK
  // as ST:
  //   %MC_JOG_ATV2(FORWARD := DRV3_JOG_INC, BACKWARD := DRV3_JOG_DEC);

// Rung 22: DRIVE_4_JOG
// DRIVE #4 JOG COMMAND
  BLK %MC_JOG_ATV3
  LD %M22                 (* DRV4_JOG_INC *)
  FORWARD
  LD %M23                 (* DRV4_JOG_DEC *)
  BACKWARD
  END_BLK
  // as ST:
  //   %MC_JOG_ATV3(FORWARD := DRV4_JOG_INC, BACKWARD := DRV4_JOG_DEC);

POU DRIVE_MOVE
  (* SectionNumber=0 *)

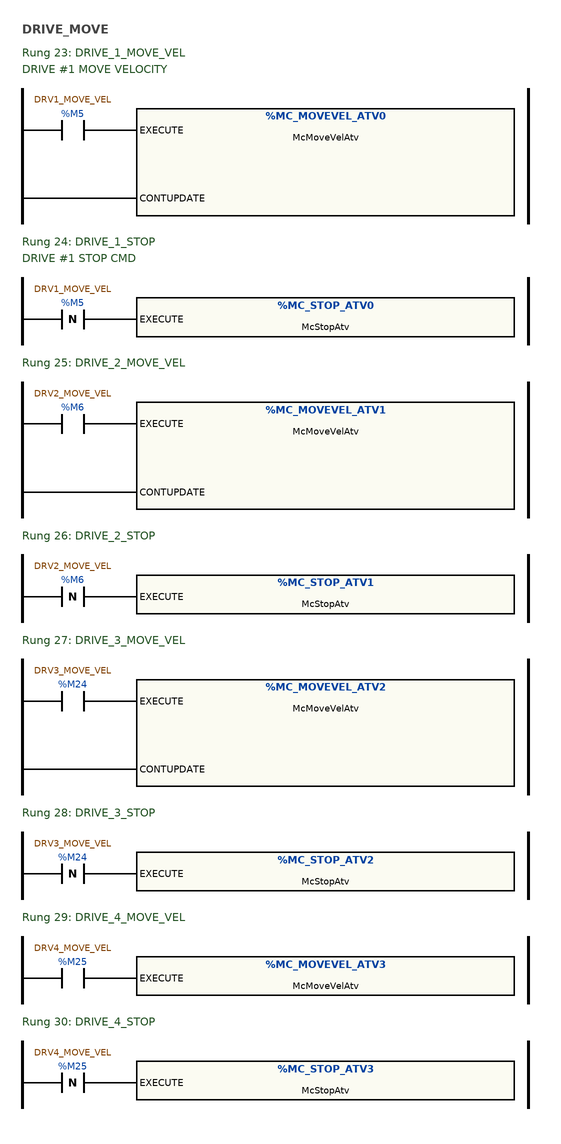

// Rung 23: DRIVE_1_MOVE_VEL
// DRIVE #1 MOVE VELOCITY
  BLK %MC_MOVEVEL_ATV0
  LD %M5                  (* DRV1_MOVE_VEL *)
  EXECUTE
  LD 1
  CONTUPDATE
  END_BLK
  // as ST:
  //   %MC_MOVEVEL_ATV0(EXECUTE := DRV1_MOVE_VEL, CONTUPDATE := TRUE);

// Rung 24: DRIVE_1_STOP
// DRIVE #1 STOP CMD
  BLK %MC_STOP_ATV0
  LDF %M5                 (* DRV1_MOVE_VEL *)
  EXECUTE
  END_BLK
  // as ST:
  //   %MC_STOP_ATV0(EXECUTE := FALLING(DRV1_MOVE_VEL));

// Rung 25: DRIVE_2_MOVE_VEL
  BLK %MC_MOVEVEL_ATV1
  LD %M6                  (* DRV2_MOVE_VEL *)
  EXECUTE
  LD 1
  CONTUPDATE
  END_BLK
  // as ST:
  //   %MC_MOVEVEL_ATV1(EXECUTE := DRV2_MOVE_VEL, CONTUPDATE := TRUE);

// Rung 26: DRIVE_2_STOP
  BLK %MC_STOP_ATV1
  LDF %M6                 (* DRV2_MOVE_VEL *)
  EXECUTE
  END_BLK
  // as ST:
  //   %MC_STOP_ATV1(EXECUTE := FALLING(DRV2_MOVE_VEL));

// Rung 27: DRIVE_3_MOVE_VEL
  BLK %MC_MOVEVEL_ATV2
  LD %M24                 (* DRV3_MOVE_VEL *)
  EXECUTE
  LD 1
  CONTUPDATE
  END_BLK
  // as ST:
  //   %MC_MOVEVEL_ATV2(EXECUTE := DRV3_MOVE_VEL, CONTUPDATE := TRUE);

// Rung 28: DRIVE_3_STOP
  BLK %MC_STOP_ATV2
  LDF %M24                (* DRV3_MOVE_VEL *)
  EXECUTE
  END_BLK
  // as ST:
  //   %MC_STOP_ATV2(EXECUTE := FALLING(DRV3_MOVE_VEL));

// Rung 29: DRIVE_4_MOVE_VEL
  BLK %MC_MOVEVEL_ATV3
  LD %M25                 (* DRV4_MOVE_VEL *)
  EXECUTE
  END_BLK
  // as ST:
  //   %MC_MOVEVEL_ATV3(EXECUTE := DRV4_MOVE_VEL);

// Rung 30: DRIVE_4_STOP
  BLK %MC_STOP_ATV3
  LDF %M25                (* DRV4_MOVE_VEL *)
  EXECUTE
  END_BLK
  // as ST:
  //   %MC_STOP_ATV3(EXECUTE := FALLING(DRV4_MOVE_VEL));

POU DRIVE_STATUS
  (* SectionNumber=0 *)

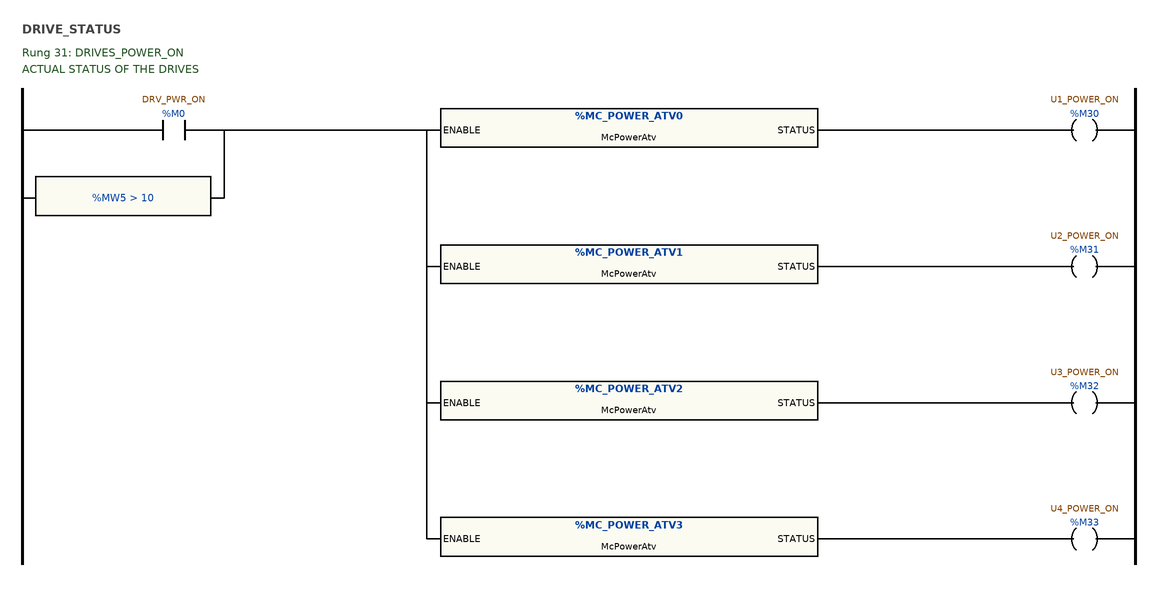

// Rung 31: DRIVES_POWER_ON
// ACTUAL STATUS OF THE DRIVES
  LD 1
  MULTIFB
  LD 1
  AND %M0                 (* DRV_PWR_ON *)
  OR [ %MW5 > 10 ]        (* FSM *)
  ST %MW2009:X0
  BLK %MC_POWER_ATV0
  LD %MW2009:X0
  ENABLE
  OUT_BLK
  LD STATUS
  ST %M30                 (* U1_POWER_ON *)
  END_BLK
  BLK %MC_POWER_ATV1
  LD %MW2009:X0
  ENABLE
  OUT_BLK
  LD STATUS
  ST %M31                 (* U2_POWER_ON *)
  END_BLK
  BLK %MC_POWER_ATV2
  LD %MW2009:X0
  ENABLE
  OUT_BLK
  LD STATUS
  ST %M32                 (* U3_POWER_ON *)
  END_BLK
  BLK %MC_POWER_ATV3
  LD %MW2009:X0
  ENABLE
  OUT_BLK
  LD STATUS
  ST %M33                 (* U4_POWER_ON *)
  END_BLK
  MULTIFB
  // as ST:
  //   %MC_POWER_ATV0(ENABLE := DRV_PWR_ON OR FSM > 10);
  //   U1_POWER_ON := %MC_POWER_ATV0.STATUS;
  //   %MC_POWER_ATV1(ENABLE := DRV_PWR_ON OR FSM > 10);
  //   U2_POWER_ON := %MC_POWER_ATV1.STATUS;
  //   %MC_POWER_ATV2(ENABLE := DRV_PWR_ON OR FSM > 10);
  //   U3_POWER_ON := %MC_POWER_ATV2.STATUS;
  //   %MC_POWER_ATV3(ENABLE := DRV_PWR_ON OR FSM > 10);
  //   U4_POWER_ON := %MC_POWER_ATV3.STATUS;

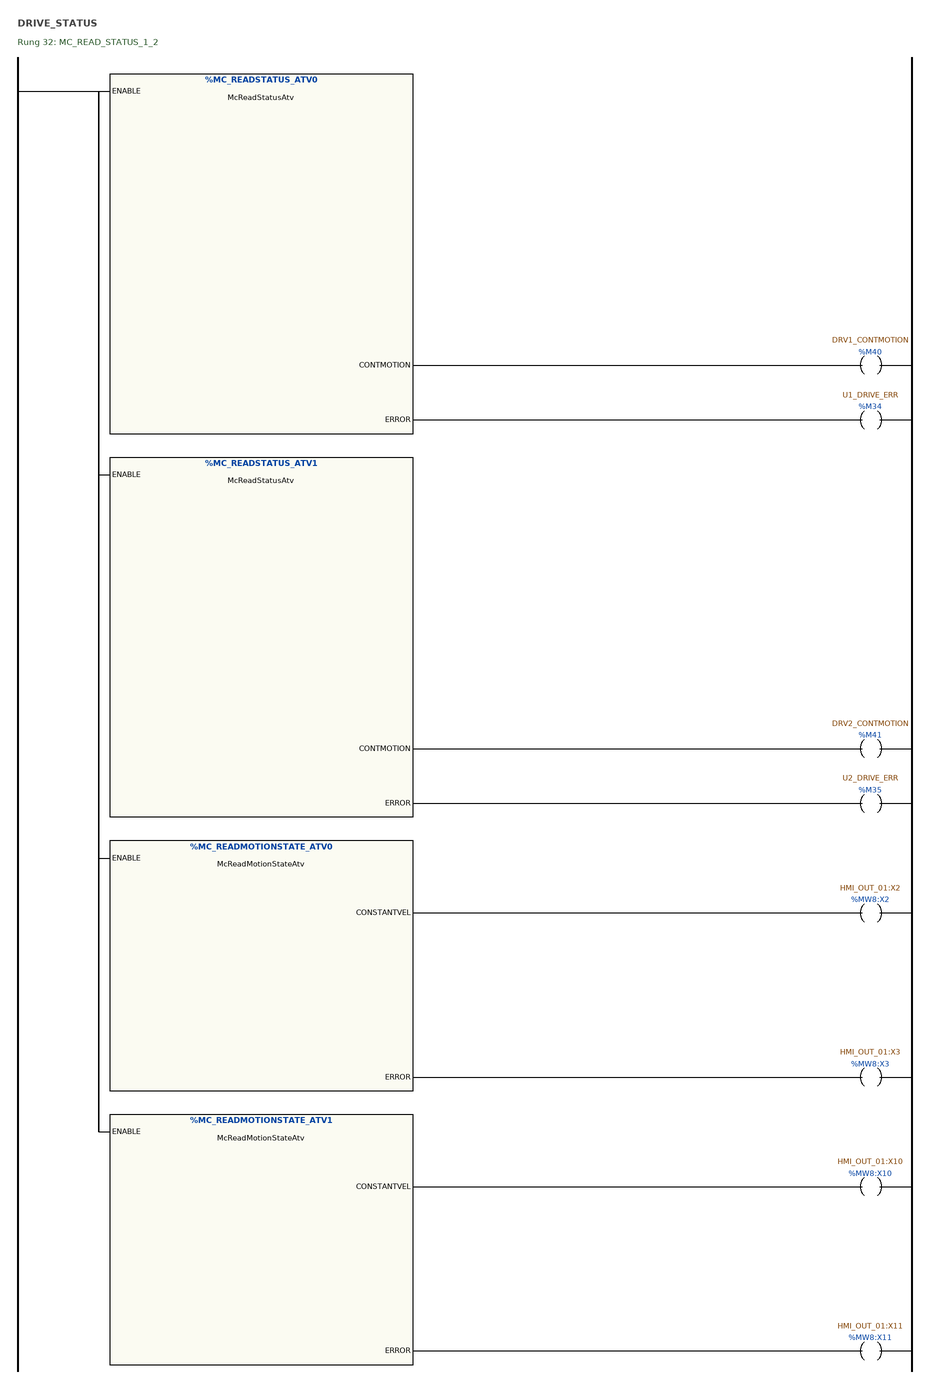

// Rung 32: MC_READ_STATUS_1_2
  LD 1
  MULTIFB
  LD 1
  ST %MW2009:X0
  BLK %MC_READSTATUS_ATV0
  LD %MW2009:X0
  ENABLE
  OUT_BLK
  LD CONTMOTION
  ST %M40                 (* DRV1_CONTMOTION *)
  LD ERROR
  ST %M34                 (* U1_DRIVE_ERR *)
  END_BLK
  BLK %MC_READSTATUS_ATV1
  LD %MW2009:X0
  ENABLE
  OUT_BLK
  LD CONTMOTION
  ST %M41                 (* DRV2_CONTMOTION *)
  LD ERROR
  ST %M35                 (* U2_DRIVE_ERR *)
  END_BLK
  BLK %MC_READMOTIONSTATE_ATV0
  LD %MW2009:X0
  ENABLE
  OUT_BLK
  LD CONSTANTVEL
  ST %MW8:X2              (* HMI_OUT_01 *)
  LD ERROR
  ST %MW8:X3              (* HMI_OUT_01 *)
  END_BLK
  BLK %MC_READMOTIONSTATE_ATV1
  LD %MW2009:X0
  ENABLE
  OUT_BLK
  LD CONSTANTVEL
  ST %MW8:X10             (* HMI_OUT_01 *)
  LD ERROR
  ST %MW8:X11             (* HMI_OUT_01 *)
  END_BLK
  MULTIFB
  // as ST:
  //   %MC_READSTATUS_ATV0(ENABLE := TRUE);
  //   DRV1_CONTMOTION := %MC_READSTATUS_ATV0.CONTMOTION;
  //   U1_DRIVE_ERR := %MC_READSTATUS_ATV0.ERROR;
  //   %MC_READSTATUS_ATV1(ENABLE := TRUE);
  //   DRV2_CONTMOTION := %MC_READSTATUS_ATV1.CONTMOTION;
  //   U2_DRIVE_ERR := %MC_READSTATUS_ATV1.ERROR;
  //   %MC_READMOTIONSTATE_ATV0(ENABLE := TRUE);
  //   HMI_OUT_01:X2 := %MC_READMOTIONSTATE_ATV0.CONSTANTVEL;
  //   HMI_OUT_01:X3 := %MC_READMOTIONSTATE_ATV0.ERROR;
  //   %MC_READMOTIONSTATE_ATV1(ENABLE := TRUE);
  //   HMI_OUT_01:X10 := %MC_READMOTIONSTATE_ATV1.CONSTANTVEL;
  //   HMI_OUT_01:X11 := %MC_READMOTIONSTATE_ATV1.ERROR;

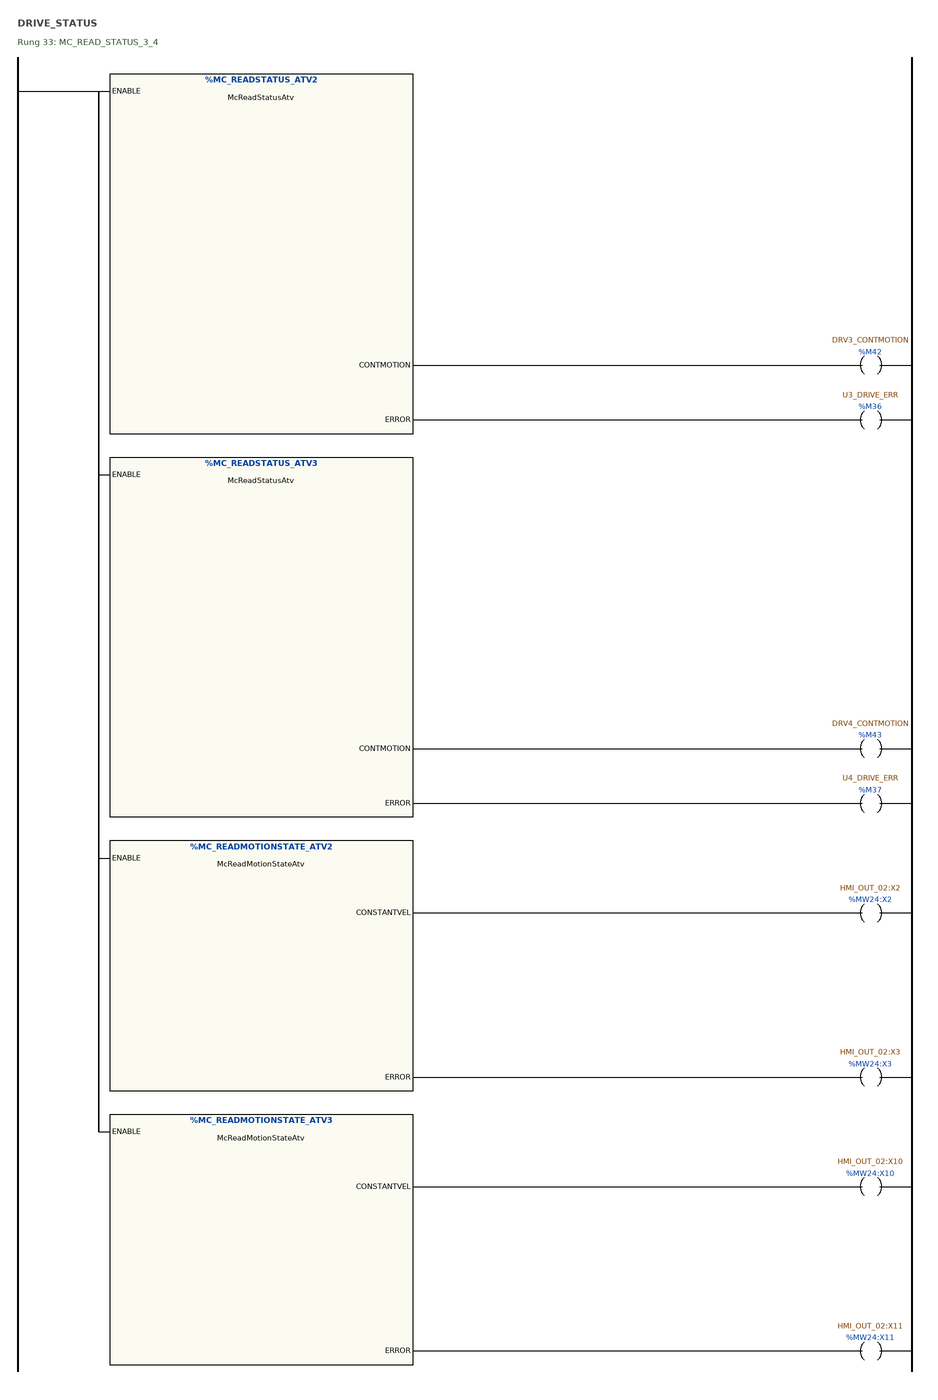

// Rung 33: MC_READ_STATUS_3_4
  LD 1
  MULTIFB
  LD 1
  ST %MW2009:X0
  BLK %MC_READSTATUS_ATV2
  LD %MW2009:X0
  ENABLE
  OUT_BLK
  LD CONTMOTION
  ST %M42                 (* DRV3_CONTMOTION *)
  LD ERROR
  ST %M36                 (* U3_DRIVE_ERR *)
  END_BLK
  BLK %MC_READSTATUS_ATV3
  LD %MW2009:X0
  ENABLE
  OUT_BLK
  LD CONTMOTION
  ST %M43                 (* DRV4_CONTMOTION *)
  LD ERROR
  ST %M37                 (* U4_DRIVE_ERR *)
  END_BLK
  BLK %MC_READMOTIONSTATE_ATV2
  LD %MW2009:X0
  ENABLE
  OUT_BLK
  LD CONSTANTVEL
  ST %MW24:X2             (* HMI_OUT_02 *)
  LD ERROR
  ST %MW24:X3             (* HMI_OUT_02 *)
  END_BLK
  BLK %MC_READMOTIONSTATE_ATV3
  LD %MW2009:X0
  ENABLE
  OUT_BLK
  LD CONSTANTVEL
  ST %MW24:X10            (* HMI_OUT_02 *)
  LD ERROR
  ST %MW24:X11            (* HMI_OUT_02 *)
  END_BLK
  MULTIFB
  // as ST:
  //   %MC_READSTATUS_ATV2(ENABLE := TRUE);
  //   DRV3_CONTMOTION := %MC_READSTATUS_ATV2.CONTMOTION;
  //   U3_DRIVE_ERR := %MC_READSTATUS_ATV2.ERROR;
  //   %MC_READSTATUS_ATV3(ENABLE := TRUE);
  //   DRV4_CONTMOTION := %MC_READSTATUS_ATV3.CONTMOTION;
  //   U4_DRIVE_ERR := %MC_READSTATUS_ATV3.ERROR;
  //   %MC_READMOTIONSTATE_ATV2(ENABLE := TRUE);
  //   HMI_OUT_02:X2 := %MC_READMOTIONSTATE_ATV2.CONSTANTVEL;
  //   HMI_OUT_02:X3 := %MC_READMOTIONSTATE_ATV2.ERROR;
  //   %MC_READMOTIONSTATE_ATV3(ENABLE := TRUE);
  //   HMI_OUT_02:X10 := %MC_READMOTIONSTATE_ATV3.CONSTANTVEL;
  //   HMI_OUT_02:X11 := %MC_READMOTIONSTATE_ATV3.ERROR;

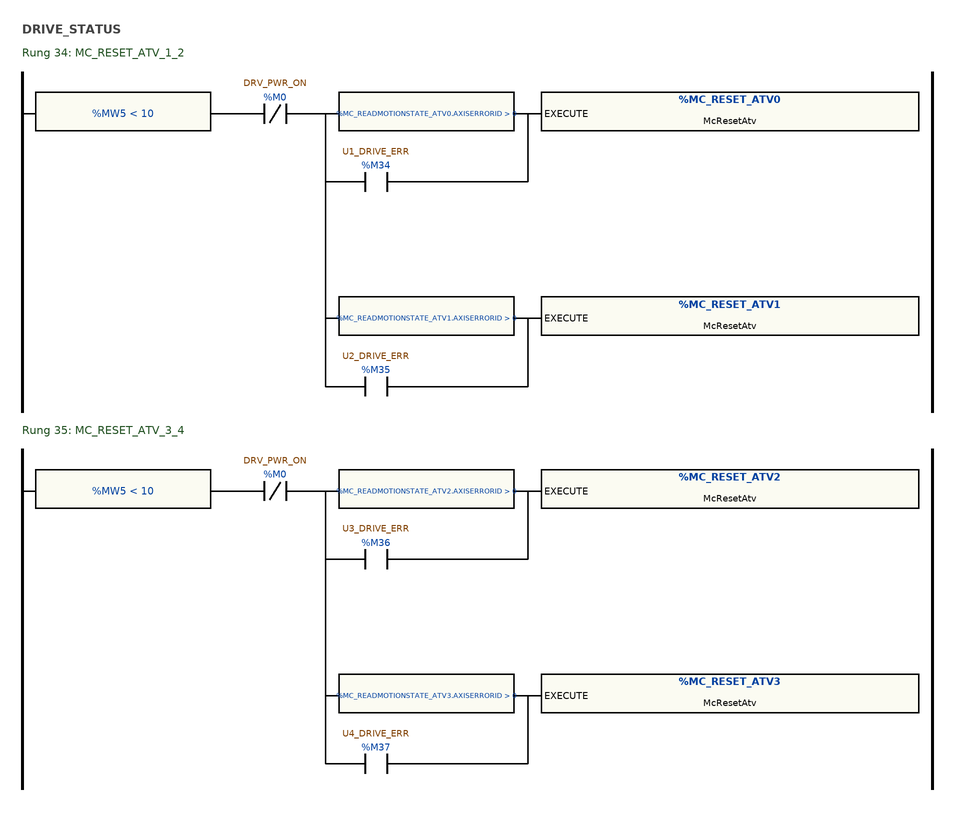

// Rung 34: MC_RESET_ATV_1_2
  LD 1
  MULTIFB
  LD 1
  AND [ %MW5 < 10 ]       (* FSM *)
  ANDN %M0                (* DRV_PWR_ON *)
  ST %MW2009:X0
  BLK %MC_RESET_ATV0
  LD %MW2009:X0
  AND( [ %MC_READMOTIONSTATE_ATV0.AXISERRORID > 0 ]
  OR %M34                 (* U1_DRIVE_ERR *)
  )
  EXECUTE
  END_BLK
  BLK %MC_RESET_ATV1
  LD %MW2009:X0
  AND( [ %MC_READMOTIONSTATE_ATV1.AXISERRORID > 0 ]
  OR %M35                 (* U2_DRIVE_ERR *)
  )
  EXECUTE
  END_BLK
  MULTIFB
  // as ST:
  //   %MC_RESET_ATV0(EXECUTE := FSM < 10 AND NOT DRV_PWR_ON AND (%MC_READMOTIONSTATE_ATV0.AXISERRORID > 0 OR U1_DRIVE_ERR));
  //   %MC_RESET_ATV1(EXECUTE := FSM < 10 AND NOT DRV_PWR_ON AND (%MC_READMOTIONSTATE_ATV1.AXISERRORID > 0 OR U2_DRIVE_ERR));

// Rung 35: MC_RESET_ATV_3_4
  LD 1
  MULTIFB
  LD 1
  AND [ %MW5 < 10 ]       (* FSM *)
  ANDN %M0                (* DRV_PWR_ON *)
  ST %MW2009:X0
  BLK %MC_RESET_ATV2
  LD %MW2009:X0
  AND( [ %MC_READMOTIONSTATE_ATV2.AXISERRORID > 0 ]
  OR %M36                 (* U3_DRIVE_ERR *)
  )
  EXECUTE
  END_BLK
  BLK %MC_RESET_ATV3
  LD %MW2009:X0
  AND( [ %MC_READMOTIONSTATE_ATV3.AXISERRORID > 0 ]
  OR %M37                 (* U4_DRIVE_ERR *)
  )
  EXECUTE
  END_BLK
  MULTIFB
  // as ST:
  //   %MC_RESET_ATV2(EXECUTE := FSM < 10 AND NOT DRV_PWR_ON AND (%MC_READMOTIONSTATE_ATV2.AXISERRORID > 0 OR U3_DRIVE_ERR));
  //   %MC_RESET_ATV3(EXECUTE := FSM < 10 AND NOT DRV_PWR_ON AND (%MC_READMOTIONSTATE_ATV3.AXISERRORID > 0 OR U4_DRIVE_ERR));
